// TIA Portal V18 export
DATA_BLOCK "NG_DB"   // DB2901
// stored: AutoNumber false, InstanceOfName NG, InstanceOfType FB
"NG"
   // VAR
   //    NG_L_1 : "NGStatus";
   //    NG_L_2 { S7_SetPoint := 'True'} : "NGStatus";
   //    NG_L_3 { S7_SetPoint := 'True'} : "NGStatus";
   //    NG_UL_1 { S7_SetPoint := 'True'} : "NGStatus";
   //    NG_UL_2 { S7_SetPoint := 'True'} : "NGStatus";
   //    NG_UL_3 { S7_SetPoint := 'True'} : "NGStatus";
   // END_VAR
BEGIN
END_DATA_BLOCK
